{attribute 'c++_compatible'}
FUNCTION_BLOCK JsonSaxHandler IMPLEMENTS ITcJsonSaxHandler
VAR_INPUT
END_VAR
VAR_OUTPUT
END_VAR
VAR
	(* Values from JSON - written by callback methods *)	  
	keystate			: INT := 0;
	label				: STRING(255);
	tempkey				: STRING(255);
	
	(* State machine variables *)
	//eState				: E_JsonStates;
	
	(* Indicators if an expected property has been found in JSON *)
	bStartObjectFound 	: BOOL;
	bEndObjectFound		: BOOL;
	
	(* Error indicators *)
	bError				: BOOL;
	sErrorMsg			: STRING(255);
END_VAR

IF bError THEN
	sErrorMsg := 'JSON message does not equal expected format';
END_IF

{attribute 'show'}
{attribute 'c++_compatible'}
{attribute 'minimal_input_size' := '4'}
{attribute 'pack_mode' := '4'}
METHOD OnBool : HRESULT
VAR_INPUT
	value	: BOOL;
END_VAR

	IF label = 'MOTION/CTR' THEN
		IF tempkey = 'CMDADD' THEN
			GVL_MOTION.EXT_CTR.CMDADD := value;
		ELSIF tempkey = 'CMDCLR' THEN
			GVL_MOTION.EXT_CTR.CMDCLR := value;
		ELSIF tempkey = 'CMDSCRIPTDEL' THEN
			GVL_MOTION.EXT_CTR.CMDSCRIPTDEL := value;	
		ELSIF tempkey = 'CMDDEL' THEN
			GVL_MOTION.EXT_CTR.CMDDEL := value;	
		ELSIF tempkey = 'CMDRUN' THEN
			GVL_MOTION.EXT_CTR.CMDRUN := value;
		ELSIF tempkey = 'CMDLOOP' THEN
			GVL_MOTION.EXT_CTR.CMDLOOP := value;	
		ELSIF tempkey = 'CMDHOME' THEN
			GVL_MOTION.EXT_CTR.CMDHOME := value;
		ELSIF tempkey = 'CMDHOMEX' THEN
			GVL_MOTION.EXT_CTR.CMDHOMEX := value;
		ELSIF tempkey = 'CMDHOMEY' THEN
			GVL_MOTION.EXT_CTR.CMDHOMEY := value;
		ELSIF tempkey = 'CMDHOMEZ' THEN
			GVL_MOTION.EXT_CTR.CMDHOMEZ := value;	
		ELSIF tempkey = 'CMDCOUPLE' THEN
			GVL_MOTION.EXT_CTR.CMDCOUPLE := value;					
		ELSIF tempkey = 'STOP' THEN
			GVL_MOTION.EXT_CTR.STOP := value;	
		ELSIF tempkey = 'AXESEN' THEN
			GVL_MOTION.EXT_CTR.AXESEN := value;		
		ELSIF tempkey = 'AXESRESET' THEN
			GVL_MOTION.EXT_CTR.AXESRESET := value;	
		ELSIF tempkey = 'CMDSCRIPTWRITE' THEN
			GVL_MOTION.EXT_CTR.CMDSCRIPTWRITE := value;
		ELSIF tempkey = 'CMDSCRIPTREAD' THEN
			GVL_MOTION.EXT_CTR.CMDSCRIPTREAD := value;	
		ELSIF tempkey = 'CMDREQLIST' THEN
			GVL_MOTION.EXT_CTR.CMDREQLIST := value;
		ELSIF tempkey = 'CMDREQSCRIPT' THEN
			GVL_MOTION.EXT_CTR.CMDREQSCRIPT := value;	
		ELSIF tempkey = 'XJOGFW' THEN
			GVL_MOTION.EXT_CTR.XJOGFW := value;
		ELSIF tempkey = 'XJOGBW' THEN
			GVL_MOTION.EXT_CTR.XJOGBW := value;
		ELSIF tempkey = 'YJOGFW' THEN
			GVL_MOTION.EXT_CTR.YJOGFW := value;
		ELSIF tempkey = 'YJOGBW' THEN
			GVL_MOTION.EXT_CTR.YJOGBW := value;
		ELSIF tempkey = 'ZJOGFW' THEN
			GVL_MOTION.EXT_CTR.ZJOGFW := value;
		ELSIF tempkey = 'ZJOGBW' THEN
			GVL_MOTION.EXT_CTR.ZJOGBW := value;	
		ELSIF tempkey = 'SETXPOS' THEN
			GVL_MOTION.EXT_CTR.SETXPOS := value;
		ELSIF tempkey = 'SETYPOS' THEN
			GVL_MOTION.EXT_CTR.SETYPOS := value;
		ELSIF tempkey = 'SETZPOS' THEN
			GVL_MOTION.EXT_CTR.SETZPOS := value;	
		ELSIF tempkey = 'BASINCTR' THEN
			GVL_MOTION.EXT_CTR.BASINCTR := value;
		ELSIF tempkey = 'BRAKEREL' THEN
			GVL_MOTION.EXT_CTR.BRAKEREL := value;
		ELSIF tempkey = 'MOVEX' THEN
			GVL_MOTION.EXT_CTR.MOVEX := value;
		ELSIF tempkey = 'MOVEY' THEN
			GVL_MOTION.EXT_CTR.MOVEY := value;
		ELSIF tempkey = 'MOVEZ' THEN
			GVL_MOTION.EXT_CTR.MOVEZ := value;							
		END_IF		
	ELSIF label = 'MOTION/HB' THEN
		IF tempkey = 'HEARTBEAT' THEN
			GVL_MOTION.HB.HEARTBEAT := value;
		END_IF	
// 	ELSIF label = 'DAQ/CTR' THEN
// 		IF tempkey = 'CMDDATACLR' THEN
// 			GVL_DAQ.TEST_CTR.CMDDATACLR := value;	
// 		ELSIF tempkey = 'CMDDATAAPEND' THEN
// 			GVL_DAQ.TEST_CTR.CMDDATAAPEND := value;
// 		ELSIF tempkey = 'CMDDATAWRITE' THEN
// 			GVL_DAQ.TEST_CTR.CMDDATAWRITE := value;
// 		END_IF	
// 	ELSIF label = 'MOTION/INSTR_BUFFER' THEN
// 		IF tempkey = 'Acq_Keyence' THEN
// 			GVL_MOTION.TestBuffer.Acq_Keyence := value;
// 		ELSIF tempkey = 'Acq_Massa' THEN
// 			GVL_MOTION.TestBuffer.Acq_Massa := value;
// 		ELSIF tempkey = 'Acq_Sonar' THEN
// 			GVL_MOTION.TestBuffer.Acq_Sonar := value;
// 		END_IF	
		
	END_IF
END_METHOD

{attribute 'show'}
{attribute 'c++_compatible'}
{attribute 'minimal_input_size' := '4'}
{attribute 'pack_mode' := '4'}
METHOD OnDint : HRESULT
VAR_INPUT
	value	: DINT;
END_VAR
// := value;
END_METHOD

{attribute 'show'}
{attribute 'c++_compatible'}
{attribute 'minimal_input_size' := '4'}
{attribute 'pack_mode' := '4'}
METHOD OnEndArray : HRESULT
VAR_INPUT
	elementCount	: UDINT;
END_VAR
END_METHOD

{attribute 'show'}
{attribute 'c++_compatible'}
{attribute 'minimal_input_size' := '4'}
{attribute 'pack_mode' := '4'}
METHOD OnEndObject : HRESULT
VAR_INPUT
	memberCount	: UDINT;
END_VAR
// IF (eState = 100) THEN
// 	bEndObjectFound := TRUE;
// 	eState := 110;  
// 	ELSE
// 		IF (eState = 110) THEN
// 			bEndObjectFound := TRUE;
// 			eState := 120;
// 		ELSE
// 			bError := TRUE;  
// 	  END_IF			
// END_IF

//keystate := keystate - 1;
END_METHOD

{attribute 'show'}
{attribute 'c++_compatible'}
{attribute 'minimal_input_size' := '4'}
{attribute 'pack_mode' := '4'}
METHOD OnKey : HRESULT
VAR_IN_OUT CONSTANT
	key	: STRING;
END_VAR
VAR_INPUT
	len	: UDINT;
END_VAR


// IF keystate = 1 THEN
// 	label := key;
// ELSIF keystate > 1 THEN
// 	tempkey	:= key;
// 	bStartObjectFound := FALSE;
// END_IF

tempkey	:= key;
END_METHOD

{attribute 'show'}
{attribute 'c++_compatible'}
{attribute 'minimal_input_size' := '4'}
{attribute 'pack_mode' := '4'}
METHOD OnLint : HRESULT
VAR_INPUT
	value	: LINT;
END_VAR
END_METHOD

{attribute 'show'}
{attribute 'c++_compatible'}
{attribute 'minimal_input_size' := '4'}
{attribute 'pack_mode' := '4'}
METHOD OnLreal : HRESULT
VAR_INPUT
	value	: LREAL;
END_VAR
// IF (eState = 70) THEN
// 	bSensor1ValueFound := TRUE;
// 	Sensor1 := value;
// 	eState := 80;
// ELSE
// 	bError := TRUE;
// 	OnLreal := S_FALSE;
// END_IF

	IF label = 'MOTION/INSTR_BUFFER' THEN
		IF tempkey = 'SetXPosition' THEN
			GVL_MOTION.InstructionBuffer.SetXPosition		:= value;
		ELSIF tempkey = 'SetYPosition' THEN
			GVL_MOTION.InstructionBuffer.SetYPosition		:= value;
		ELSIF tempkey = 'SetZPosition' THEN
			GVL_MOTION.InstructionBuffer.SetZPosition		:= value;	
		END_IF
	ELSIF label = 'MOTION/CTR' THEN	
		IF tempkey = 'POSX' THEN
			GVL_MOTION.EXT_CTR.POSX		:= value;
		ELSIF tempkey = 'POSY' THEN
			GVL_MOTION.EXT_CTR.POSY		:= value;
		ELSIF tempkey = 'POSZ' THEN
			GVL_MOTION.EXT_CTR.POSZ		:= value;	
		END_IF
	END_IF
END_METHOD

{attribute 'show'}
{attribute 'c++_compatible'}
{attribute 'minimal_input_size' := '4'}
{attribute 'pack_mode' := '4'}
METHOD OnNull : HRESULT
END_METHOD

{attribute 'show'}
{attribute 'c++_compatible'}
{attribute 'minimal_input_size' := '4'}
{attribute 'pack_mode' := '4'}
METHOD OnRawNumber : HRESULT
VAR_IN_OUT CONSTANT
	value	: STRING;
END_VAR
VAR_INPUT
	len	: UDINT;
END_VAR
END_METHOD

{attribute 'show'}
{attribute 'c++_compatible'}
{attribute 'minimal_input_size' := '4'}
{attribute 'pack_mode' := '4'}
METHOD OnStartArray : HRESULT
END_METHOD

{attribute 'show'}
{attribute 'c++_compatible'}
{attribute 'minimal_input_size' := '4'}
{attribute 'pack_mode' := '4'}
METHOD OnStartObject : HRESULT

//keystate := keystate + 1;
label := GVL_MOTION.TopicRcv;
bStartObjectFound := TRUE;
END_METHOD

{attribute 'show'}
{attribute 'c++_compatible'}
{attribute 'minimal_input_size' := '4'}
{attribute 'pack_mode' := '4'}
METHOD OnString : HRESULT
VAR_IN_OUT CONSTANT
	value	: STRING;
END_VAR
VAR_INPUT
	len	: UDINT;
END_VAR
// IF (eState = 50) THEN
// 	bTimestampValueFound := TRUE;
// 	STRNCPY(pDst:=ADR(sTimestamp), pSrc:=ADR(value), nDstSize:=SIZEOF(sTimestamp));
// 	eState := 60;
// ELSE
// 	bError := TRUE;
// 	OnString := S_FALSE;
// END_IF

	IF label = 'MOTION/INSTR_BUFFER' THEN
		IF tempkey = 'Comment' THEN
			GVL_MOTION.InstructionBuffer.Comment		:= value;
		END_IF
	ELSIF label = 'MOTION/CTR' THEN
		IF tempkey = 'SCRIPTNAME' THEN
			GVL_MOTION.EXT_CTR.SCRIPTNAME		:= value;
		END_IF	
	END_IF
END_METHOD

{attribute 'show'}
{attribute 'c++_compatible'}
{attribute 'minimal_input_size' := '4'}
{attribute 'pack_mode' := '4'}
METHOD OnUdint : HRESULT
VAR_INPUT
	value		:UDINT;
END_VAR
VAR
	//temptime	:TIME;
END_VAR
// IF (eState = 90) THEN
// 	bSensor2ValueFound := TRUE;
// 	Sensor2 := value;
// 	eState := 100;
// ELSE
// 	bError := TRUE;TO_TIME
// 	OnUdint := S_FALSE;
// END_IF

	IF label = 'MOTION/INSTR_BUFFER' THEN
		IF tempkey = 'MotionCommand' THEN
			GVL_MOTION.InstructionBuffer.MotionCommand		:= UDINT_TO_INT(value);
// 		ELSIF tempkey = 'zType' THEN
// 			GVL_MOTION.TestBuffer.zType				:= UDINT_TO_INT(value);
// 		ELSIF tempkey = 'DataTrigger' THEN
// 			GVL_MOTION.TestBuffer.DataTrigger		:= UDINT_TO_INT(value);	
		ELSIF tempkey = 'SetXPosition' THEN
			GVL_MOTION.InstructionBuffer.SetXPosition		:= UDINT_TO_INT(value);
		ELSIF tempkey = 'SetXVelocity' THEN
			GVL_MOTION.InstructionBuffer.SetXVelocity		:= UDINT_TO_INT(value);
		ELSIF tempkey = 'SetXAccel' THEN
			GVL_MOTION.InstructionBuffer.SetXAccel			:= UDINT_TO_INT(value);
		ELSIF tempkey = 'SetYPosition' THEN
			GVL_MOTION.InstructionBuffer.SetYPosition		:= UDINT_TO_INT(value);
		ELSIF tempkey = 'SetYVelocity' THEN
			GVL_MOTION.InstructionBuffer.SetYVelocity		:= UDINT_TO_INT(value);
		ELSIF tempkey = 'SetYAccel' THEN
			GVL_MOTION.InstructionBuffer.SetYAccel			:= UDINT_TO_INT(value);
		ELSIF tempkey = 'SetZPosition' THEN
			GVL_MOTION.InstructionBuffer.SetZPosition		:= UDINT_TO_INT(value);
		ELSIF tempkey = 'SetZVelocity' THEN
			GVL_MOTION.InstructionBuffer.SetZVelocity		:= UDINT_TO_INT(value);			
		ELSIF tempkey = 'PauseTime' THEN
			//temptime := TIME#1MS * value;
			GVL_MOTION.InstructionBuffer.PauseTime 		:= TIME#1MS * value;
		END_IF		
// 	ELSIF label = 'DAQ/CTR' THEN
// 		IF tempkey = 'DAQRES' THEN
// 			GVL_DAQ.TEST_CTR.DAQRES				:= UDINT_TO_INT(value);
// 		END_IF	
	ELSIF label = 'MOTION/CTR' THEN	
		IF tempkey = 'SCRIPTITERATIONS' THEN 	
			GVL_MOTION.EXT_CTR.SCRIPTITERATIONS	:= UDINT_TO_INT(value);	
		END_IF
		
	END_IF
END_METHOD

{attribute 'show'}
{attribute 'c++_compatible'}
{attribute 'minimal_input_size' := '4'}
{attribute 'pack_mode' := '4'}
METHOD OnUlint : HRESULT
VAR_INPUT
	value	: ULINT;
END_VAR
END_METHOD

{attribute 'show'}
{attribute 'c++_compatible'}
{attribute 'minimal_input_size' := '4'}
{attribute 'pack_mode' := '4'}
METHOD TcAddRef : UDINT
END_METHOD

{attribute 'show'}
{attribute 'c++_compatible'}
{attribute 'minimal_input_size' := '4'}
{attribute 'pack_mode' := '4'}
METHOD TcQueryInterface : HRESULT
VAR_INPUT
	iid	: REFERENCE TO IID;
	pipItf	: POINTER TO PVOID;
END_VAR
END_METHOD

{attribute 'show'}
{attribute 'c++_compatible'}
{attribute 'minimal_input_size' := '4'}
{attribute 'pack_mode' := '4'}
METHOD TcRelease : UDINT
END_METHOD

END_FUNCTION_BLOCK

(* stored: Version 1.1.0.1, ProductVersion 3.1.4026.18
   POU JsonSaxHandler: Id {fd22ba04-0d36-44e7-a81e-c59d3ac0f333}, SpecialFunc None
   Method OnBool: Id {13455f88-e234-4d6f-b163-c3ace2d01de9}
   Method OnDint: Id {24238a66-3ba2-41ea-bb1d-dec022507274}
   Method OnEndArray: Id {1739a2d6-6bf1-4ae8-9382-66870451d46e}
   Method OnEndObject: Id {885811d0-5c76-4031-96ce-48dd447f7032}
   Method OnKey: Id {0166f13e-7ed0-43f7-a777-b23d02f1dd47}
   Method OnLint: Id {729de20b-2d3e-4125-9187-e0252a19c186}
   Method OnLreal: Id {e458c372-d873-4613-adb7-f607191d076c}
   Method OnNull: Id {65642340-6997-4108-83d9-c8813a05825e}
   Method OnRawNumber: Id {f9737890-9bac-4333-b9b2-37d74169c053}
   Method OnStartArray: Id {655fbaa9-4596-43be-8c13-3d5daaf75b5e}
   Method OnStartObject: Id {9da87a42-4b27-47bf-b4fc-3d1a5b5e45be}
   Method OnString: Id {1c13bada-871d-4b30-bee1-08ea70607c6f}
   Method OnUdint: Id {296ac94a-f1f7-4890-a4b8-5d9fd3b55ce6}
   Method OnUlint: Id {3d01b1c5-c02d-481b-a604-269325783bc9}
   Method TcAddRef: Id {ed9db009-45ee-459b-bd3c-e6eebd2276ca}
   Method TcQueryInterface: Id {bf125ab6-3d6a-4df3-b162-942f3b1feb6f}
   Method TcRelease: Id {f07919cf-792d-4887-afc7-1c9d1066ed11} *)
